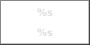
VISUALIZATION F_DiagramState  // 90x45
VAR_IN_OUT
	stStateInfo		: ST_MCHMIPrepareScreen_06_XX_State;
END_VAR
    Rectangle (0,0 90x45), colour variable: stStateInfo.dwBackgroud
        p1271844420: stStateInfo.iWidthFrame
    Rectangle (5,5 80x15), "%s", text variable: stStateInfo.wsNameOfState
    Rectangle (5,25 80x15), "%s", text variable: stStateInfo.sTime, invisible if: not stStateInfo.bShowTime
END_VISUALIZATION

(* stored: Version 1.1.0.1
   Visu F_DiagramState: Id {449a4647-909c-00e2-2820-61c6299bd7a1} *)
